PROGRAM MAIN
VAR
END_VAR

Taster_entprellung();
Blinker();

END_PROGRAM

(* stored: Version 1.1.0.1, ProductVersion 3.1.4022.9
   POU MAIN: Id {7dfbc7da-633e-464c-8224-cf772019737c}, SpecialFunc None *)
